FUNCTION_BLOCK PIPE_VIEW (* View of a Pipe Segment *)
  (* Standard: 61499-1; Classification: View *)
  (* Version 0.1, 2004-09-01, JHC, Rockwell Automation, Copied/Modified from CNV_VIEW *)
  (* Version 0.0, 2004-08-30, JHC, Rockwell Automation, Copied/Modified from CNV_VIEW *)
  (* Compiler header: package fb.rt.process; *)
  (* Compiler Java IBM VisualAge 3.0 *)
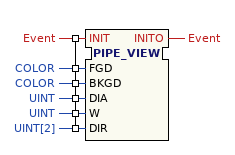
  EVENT_INPUT
    INIT WITH BKGD, DIA, W, DIR, FGD; (* Initialize *)
  END_EVENT
  EVENT_OUTPUT
    INITO; (* Initialized *)
  END_EVENT
  VAR_INPUT
    FGD : COLOR := blue; (* Foreground Color *)
    BKGD : COLOR := white; (* Background Color *)
    DIA : UINT; (* Segment side length *)
    W : UINT := 4; (* Pipe width *)
    DIR : ARRAY [0..1] OF UINT; (* [Entry,Exit]: 0=North, 1=East, 2=South, 3=West *)
  END_VAR
END_FUNCTION_BLOCK
